RoboDK station: ur5_and_table_and_indicator.rdk

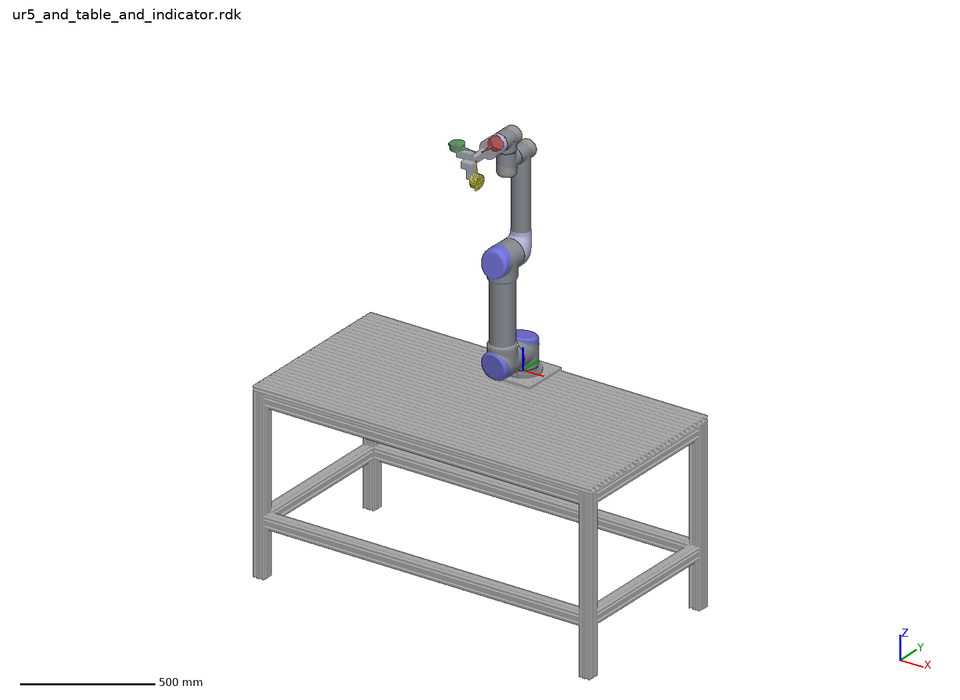
[picture v0: the station drawn from its stored meshes, robots at their saved joint values, targets as dots, program paths as lines]
Station ur5_and_table_and_indicator. Poses are relative to the parent item; angles as X-Y-Z fixed-axis rotations.
  - frame UR5 Base at (0, 0, 0) mm
    - robot UR5: 6 axes, payload 5 kg, reach 850 mm, repeatability 0.1 mm, weight 18.4 kg
        modified DH rows (alpha deg, a mm, theta deg, d mm): 0, 0, 0, 89.2; 90, 0, 180, 0; 0, 425, 0, 0; 0, 392.43, 0, 109; -90, 0, 0, 93.65; 90, 0, 180, 82
        joint limits [-360, -360, -360, -360, -360, -360] to [360, 360, 360, 360, 360, 360]; home [0, -90, 90, 0, 90, 0]; saved at [0, -90, 0, -90, 0, 0]
      - tool assembly, TCP at (0, 0, 0) mm, size 118 x 193.6 x 208.3 mm, geometry from assembly.IGS
  - object table_base_setup at (0, 0, 0) mm, rotated rx 0 ry 0 rz -90 deg, size 1524 x 762 x 800.1 mm, geometry from table_base_setup.STEP
